//==================================================================================================
//								RJM Maszyny sp. z o.o.
//									13.05.2022
//
//	Obsługa przycisku podświetlanego
//	v1.0	|| TC v 3.1.4024.22		|| - pierwsza wersja
//==================================================================================================
FUNCTION_BLOCK FB_Przycisk_NO_Podswietlany EXTENDS FB_Przycisk_NO
VAR
	bLampka							AT %Q*	: BOOL;
	
END_VAR

//==================================================================================================
//								RJM Maszyny sp. z o.o.
//									13.05.2022
//
//	Włączenie podświetlenia przycisku
//	v1.0	|| TC v 3.1.4024.22		|| - pierwsza wersja
//==================================================================================================
METHOD WlaczPodswietlenie
VAR_INPUT
END_VAR
bLampka										:= TRUE;
END_METHOD

//==================================================================================================
//								RJM Maszyny sp. z o.o.
//									13.05.2022
//
//	Wyłączenie podświetlenia przycisku
//	v1.0	|| TC v 3.1.4024.22		|| - pierwsza wersja
//==================================================================================================
METHOD WylaczPodswietlenie
VAR_INPUT
END_VAR
bLampka										:= FALSE;
END_METHOD

END_FUNCTION_BLOCK

(* stored: Version 1.1.0.1, ProductVersion 3.1.4024.11
   POU FB_Przycisk_NO_Podswietlany: Id {7c3dc557-ee66-419c-83aa-f52bffe2c58f}, SpecialFunc None
   Method WlaczPodswietlenie: Id {b05c4f20-bf3d-4224-aa6b-a763e972a792}
   Method WylaczPodswietlenie: Id {0035383d-b591-419c-8b49-be1c9d7f54ee} *)
